// TIA Portal V20 export
DATA_BLOCK "FDQ1"   // DB291
// stored: MemoryReserve 100
   VAR
      "MANIFOLD-1 SOL POWER MC ON" : Bool;
      SPARE1 : Bool;
      SPARE2 : Bool;
      SPARE3 : Bool;
      "FFU POWER MC ON 1" : Bool;
      "FFU POWER MC ON 2" : Bool;
      SPARE4 : Bool;
      SPARE5 : Bool;
   END_VAR
BEGIN
END_DATA_BLOCK
